(* CODESYS project Edificio central Gateway PLC Maestro v0.project
   Title: Sin título
   Version: 0.0.0.0
   Author: francisco.florensa

Project tree, tasks and I/O mapping:
  MyController : TM241CEC24R, Schneider Electric, order no. TM241CEC24R, version 4.0.6.18
    application Application
      task MAST (cyclic, interval 20 ms, priority 15, watchdog 100 ms x 1) calls MyPOU
      global variables GVL
      program MyPOU [LD]
      Symbols
    DI : Digital Inputs, Schneider Electric, version 4.0.6.18
        input  iwDI_IW0 : WORD  // IW0
        input  ibDI_IB1 : BYTE  // IB1
    DQ : Digital Outputs, Schneider Electric, version 4.0.6.18
        output xq_salida0 : BOOL  // QW0.Q0
        output xq_salida1 : BOOL  // QW0.Q1
        output xq_salida2 : BOOL  // QW0.Q2
        output xq_salida3 : BOOL  // QW0.Q3
        output xq_salida4 : BOOL  // QW0.Q4
        output xq_salida5 : BOOL  // QW0.Q5
        output xq_salida6 : BOOL  // QW0.Q6
        output xq_salida7 : BOOL  // QW0.Q7
        output xq_salida8 : BOOL  // QW0.Q8
        output xq_salida9 : BOOL  // QW0.Q9
        output qbDQ_QB1 : BYTE  // QB1
        unmapped channels: QW0
    Counters : Counters, Schneider Electric, version 4.0.6.18
    Pulse_Generators : Pulse Generators, Schneider Electric, version 4.0.6.18
    Cartridge_1 : Cartridge, Schneider Electric, version 4.0.6.18
    IO_Bus : IO bus - TM3, Schneider Electric, version 4.0.6.18
    COM_Bus : COM bus, Schneider Electric, version 4.0.6.18
    Ethernet_1 : Ethernet Network, Schneider Electric, version 4.0.6.18
        settings: IPAddress = [192, 168, 1, 58]; SubnetMask = [255, 255, 255, 0]; WebServer = TRUE; FTP Server = TRUE; SoMachine Protocol = TRUE; Modbus Server = TRUE; NetManage Protocol = TRUE; SNMP protocol = TRUE; Enable Routing = FALSE; WebVisu protocol = TRUE; DHCP Server Active = TRUE
    Serial_Line_1 : Serial line, Schneider Electric, version 4.0.6.18
      SoMachine_Network_Manager : SoMachine-Network Manager, Schneider Electric, version 4.0.0.2
    Serial_Line_2 : Serial line, Schneider Electric, version 4.0.6.18
      Modbus_Manager : Modbus Manager, Schneider Electric, version 4.0.0.2
    CAN_1 : CANopen bus, Schneider Electric, version 4.0.6.18
  HMISCUxA5 : HMISCUxA5, Schneider Electric, order no. HMISCUxA5, version 3.5.3.59
    application Application
      task MAST (cyclic, interval 20 ms, priority 15, watchdog 100 ms x 1) calls nothing
      global variables GVL
    HMI Application
    COM1
      SoMachine_Network_Manager1 : SoMachine-Network Manager, Schneider Electric, version 4.0.0.2
    Ethernet
      SoMachine_Network_Manager2 : SoMachine-Network Manager, Schneider Electric, version 4.0.0.2
    USB
      SoMachine_Network_Manager3 : SoMachine-Network Manager, Schneider Electric, version 4.0.0.2
    CAN
    Funciones incorporadas
      ES : ES, Schneider Electric, order no. IO, version 3.5.3.59
          input  iwES_Entrada : WORD  // In
          output qwES_Salida : WORD  // Out
      PTO_PWM : PTO_PWM, Schneider Electric, order no. PTO_PWM, version 3.5.3.59
      HSC : HSC, Schneider Electric, order no. HSC, version 3.5.3.59
  Vijeo Designer Project Container
  Vijeo Designer Project Container Data
*)

// MyController/Application/GVL
VAR_GLOBAL
	i_var0 AT %MW0:UINT;
	i_var1 AT %MW1:INT;
	i_var2 AT %MW2:INT;
	i_var3 AT %MW3:INT;
	GEN_0: GEN;
END_VAR

// HMISCUxA5/Application/GVL
VAR_GLOBAL
END_VAR

// MyController/Application/MyPOU
PROGRAM MyPOU
VAR
	WORD_AS_BIT_0: WORD_AS_BIT;
	i_sinusoidal: INT;
END_VAR

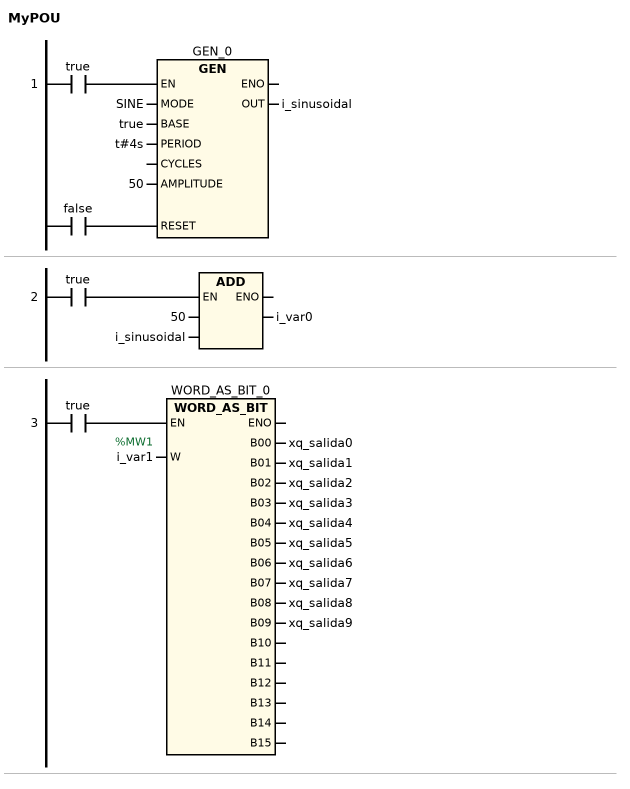
// NETWORK 1
IF true THEN
    GEN_0(MODE := SINE, BASE := true, PERIOD := t#4s, AMPLITUDE := 50, RESET := false, OUT => i_sinusoidal); // GEN
END_IF

// NETWORK 2
//   i_var0: AT %MW0
IF true THEN i_var0 := 50 + i_sinusoidal; END_IF

// NETWORK 3
//   i_var1: AT %MW1
//   xq_salida0: DQ : Salida rápida, contrafase | AT %QX0.0
//   xq_salida1: DQ : Salida rápida, contrafase | AT %QX0.1
//   xq_salida2: DQ : Salida rápida, contrafase | AT %QX0.2
//   xq_salida3: DQ : Salida rápida, contrafase | AT %QX0.3
//   xq_salida4: DQ : Salida de relé | AT %QX0.4
//   xq_salida5: DQ : Salida de relé | AT %QX0.5
//   xq_salida6: DQ : Salida de relé | AT %QX0.6
//   xq_salida7: DQ : Salida de relé | AT %QX0.7
//   xq_salida8: DQ : Salida de relé | AT %QX1.0
//   xq_salida9: DQ : Salida de relé | AT %QX1.1
IF true THEN
    WORD_AS_BIT_0(
        W := i_var1,
        B00 => xq_salida0,
        B01 => xq_salida1,
        B02 => xq_salida2,
        B03 => xq_salida3,
        B04 => xq_salida4,
        B05 => xq_salida5,
        B06 => xq_salida6,
        B07 => xq_salida7,
        B08 => xq_salida8,
        B09 => xq_salida9); // WORD_AS_BIT
END_IF

END_PROGRAM
